{attribute 'OPC.UA.DA.StructuredType' := '1'}
TYPE SNamedValue EXTENDS SValue :
STRUCT
	Name: STRING;
END_STRUCT
END_TYPE

(* stored: Version 1.1.0.1, ProductVersion 3.1.4024.9
   DUT SNamedValue: Id {3230726c-1a4b-4b2b-9eb5-b41b303f36d7} *)
